// Brief: Mounting Instrument
FUNCTION_BLOCK PUBLIC FB_SlaveCtrlMountInstru EXTENDS FB_SlaveArmCtrlBase
VAR_INPUT
END_VAR
VAR_OUTPUT
END_VAR
VAR
	// mount status
	m_mountStatus :INT := 0;
	m_J4mountStatus :INT := 0;
	
	// flag if joint is mounted
	m_jointMounted :ARRAY[1..5] OF BOOL := [5(FALSE)];
	
	// instrument mount motion range
	m_mountMotionAng :Vec5d :=[2*PI, 2*PI, 2*PI, 2*PI, 2*PI];
	
	// instrument mount direction
	m_mountDir :Vec5i :=[1, 1, 1, 1, 1];
	
	// mount motion planning
	m_jntOTG :ARRAY[1..5] OF FB_secOrdTrajFilter;
	m_instruMountVel :LREAL := 2*PI;//30* g_deg2Rad;
	m_instruMountAcc :LREAL := 2*PI;
	
	// track error threshold which indicate motor is buckled with panel
	m_maxTrackErr :LREAL := 5*g_deg2Rad;
	
	//powerbox motor stop vel
	m_stopVel :LREAL := 1*g_deg2Rad;
	
	//Joint 4 rotation angle
	rotAngleJ4 :LREAL := 323*g_deg2Rad;
	
	// joint current threshold which indicate panel is buckled with instrument
	m_maxJntCurrent :INT := 180;
	
	// command mount motion
	m_targetMountPos :Vec8d;
	
	// instrument zero position
	m_instruZeroDeviation :Mat45;
	m_PowerboxZeroPos :Mat45:=[5.75,5.75,5.75-pi,2,   5.75,5.75,5.75-pi,2,   5.75,5.75,5.75-pi,2,   5.75,5.75,5.75-pi,2];
	m_instruZeroDeviationJ4:LREAL;
	
	//instrument clamping Error
	m_Error:BOOL;
	m_ErrorID:DINT;
END_VAR

// override this function in each exact controller
METHOD PROTECTED calcCmdJntPos : BOOL
VAR_INPUT
	motionScale :LREAL;
	masterIdx :INT;
END_VAR

VAR_IN_OUT CONSTANT
	i_slaveArm :FB_SlaveArm;
	i_masterStatus :ST_MasterStatus;
END_VAR

VAR 
	i :INT;
	curJntVel :Vec8d;
	curJntPos :Vec8d;
	jntPosErr :Vec8d;
END_VAR

curJntPos := i_slaveArm.curJntPos;

CASE m_mountStatus OF
	// To lock panel with instrument
	0:
		FOR i:=1 TO 5 DO
			m_ratedCur[i+3]:=200;
			// check joint buckled with instrument
			IF ABS(i_slaveArm.filtJntCurrent[i+3])> m_maxJntCurrent THEN 
				m_jointMounted[i]:=TRUE;
				m_targetMountPos[i+3]:=curJntPos[i+3];
			END_IF
			
			// set target joint position
			IF FALSE = m_jointMounted[i] THEN
				m_targetMountPos[i+3]:=curJntPos[i+3]-m_mountMotionAng[i];
			END_IF
		END_FOR
		
		IF (m_jointMounted[1] AND m_jointMounted[2] AND m_jointMounted[3] AND m_jointMounted[4] AND m_jointMounted[5])  THEN
			IF i_slaveArm.instrument.InstruReadPara.m_InstruReadSucceed THEN//Check whether the data is read successfully
				m_mountStatus:=1;
			ELSE
				m_Error:=TRUE;
				m_ErrorID:=1;
			END_IF
		END_IF
	
	1:// The calculation deviates from the instrument zero position
		(*IF m_instruZeroDeviationJ4>PI THEN //J4
			m_instruZeroDeviation[1,4]:=m_instruZeroDeviationJ4;
		ELSE
			m_instruZeroDeviation[1,4]:=-m_instruZeroDeviationJ4;
		END_IF*)
		m_instruZeroDeviation[1,4]:=rotAngleJ4;
		
		FOR i:=1 TO 3 DO//J1-3
			m_instruZeroDeviation[1,i] := m_PowerboxZeroPos[1,i] - i_slaveArm.linkSingle[i+3] - i_slaveArm.instrument.InstruReadPara.m_InstruPos[1,i];
			IF m_instruZeroDeviation[1,i]>pi THEN
				m_instruZeroDeviation[1,i] := m_instruZeroDeviation[1,i] - 2*PI;
			ELSIF m_instruZeroDeviation[1,i]<-pi THEN
				m_instruZeroDeviation[1,i] := m_instruZeroDeviation[1,i] + 2*PI;
			END_IF
		END_FOR
		m_mountStatus :=2;
	
	
	2:// move back to zero position
	
		// set target joint position
		FOR i:=1 TO 4 DO
			m_targetMountPos[i+3]:=curJntPos[i+3] + m_instruZeroDeviation[1,i];
		END_FOR
		m_mountStatus :=3;
		
		
	3:
		m_isFinished:=TRUE;
		FOR i:=1 TO 5 DO
			IF ABS(m_targetMountPos[i+3]-curJntPos[i+3])>0.05 THEN
				m_isFinished:=FALSE;
				EXIT;
			END_IF
		END_FOR
		
		(*vecSub(m_targetMountPos,curJntPos,jntPosErr);
		IF vecNorm(jntPosErr)<GVL_SlaveControlParameters.g_jntCtrlPosTol THEN
			m_isFinished:=TRUE;
		END_IF*)
		
		(*IF  ABS(m_cmdJntPos[7]-m_targetMountPos[7])< GVL_SlaveControlParameters.g_jntCtrlPosTol THEN 
			m_targetMountPos[7]:=curJntPos[7];
		ELSIF ABS(m_cmdJntPos[7]-m_targetMountPos[7])> GVL_SlaveControlParameters.g_jntCtrlPosTol AND ABS(i_slaveArm.filtJntCurrent[7])> 80 AND i_slaveArm.curJntVel[7]<m_stopVel THEN
			
			m_targetMountPos[i+3]:=curJntPos[7]-rotAngleJ4;//direction of current
			m_mountStatus :=4;
		END_IF*)
		
	4:
		vecSub(m_targetMountPos,curJntPos,jntPosErr);
		IF vecNorm(jntPosErr)<GVL_SlaveControlParameters.g_jntCtrlPosTol THEN
			m_isFinished:=TRUE;
		END_IF
		
END_CASE

//ABS(m_cmdJntPos[7]-curJntPos[7])> m_maxTrackErr OR
//Calculate the deviation of J4 from the zero point
m_instruZeroDeviationJ4:=m_PowerboxZeroPos[1,4] - i_slaveArm.linkSingle[4+3] ;
IF m_instruZeroDeviationJ4>2*PI THEN
	m_instruZeroDeviationJ4:=m_instruZeroDeviationJ4-2*PI;
END_IF

// traj plan
FOR i:=1 TO 5 DO
	m_jntOTG[i].run(m_targetMountPos[i+3],0.0, o_cmdAcc=>m_cmdJntAcc[3+i],o_cmdVel=>m_cmdJntVel[3+i],o_cmdPos=>m_cmdJntPos[i+3]);
END_FOR
END_METHOD

METHOD PUBLIC init : BOOL
VAR_IN_OUT CONSTANT
	i_slaveArm	:FB_SlaveArm;
END_VAR
VAR_IN_OUT 
	r_slaveArmCtrlCmd :ST_SlaveArmCtrlCmds;
END_VAR

VAR
	i : INT;
END_VAR
SUPER^.Init(i_slaveArm,r_slaveArmCtrlCmd);

// check if to hold the command joint position unchanged
checkToHoldLastCmds(i_slaveArm,r_slaveArmCtrlCmd);
FOR i:=1 TO 5 DO
	m_targetMountPos[i+3]:=m_cmdJntPos[i+3];
	m_jntOTG[i].init(m_targetMountPos[i+3], 0,m_instruMountVel, m_instruMountAcc, g_slaveArmCtrlCycleTime);
	m_jointMounted[i]:=FALSE;
END_FOR

m_mountStatus:=0;
// check instrument type to get mount joint index and zero position
IF i_slaveArm.instrument.InstruReadPara.m_Instrutype <> InstruType_UNKNOWM THEN
	m_jointMounted[5]:=TRUE;

END_IF


//Update the IP and port number of the operating arm
i_slaveArm.instrument.InstruReadPara.i_ArmNetId:=GVL_SlaveMotorParameters.g_slaveArmNetID[1];
i_slaveArm.instrument.InstruReadPara.i_JointInstruAddr:=GVL_SlaveMotorParameters.g_slaveJointNetPort[1,4];

m_Error:=FALSE;
m_ErrorID:=0;
END_METHOD

END_FUNCTION_BLOCK

(* stored: Version 1.1.0.1, ProductVersion 3.1.4024.11
   POU FB_SlaveCtrlMountInstru: Id {db93de24-03af-45f5-8edb-e02a943fe1f8}, SpecialFunc None
   Method calcCmdJntPos: Id {106b8ce6-26fa-4bca-bfc9-20f8cdf00f0e}
   Method init: Id {85ccbdcb-d27d-4162-a6ec-e8e93d30dbc6} *)
